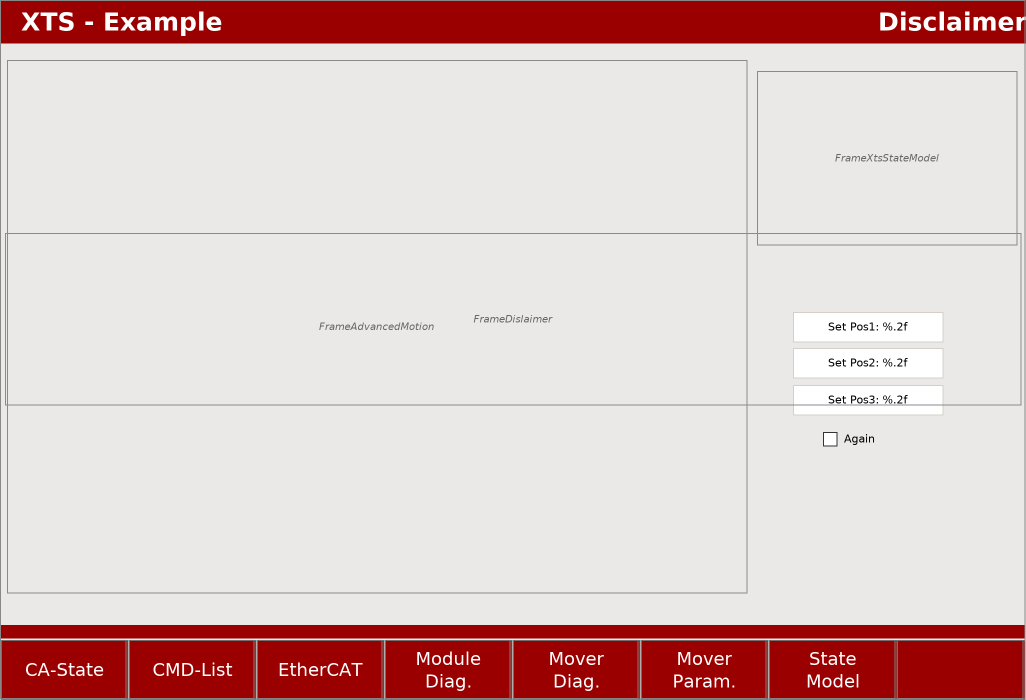
VISUALIZATION FrameVisuSimpelCaExample  // 1026x700
VAR_IN_OUT
	
	stVisuIO		: ST_VisuExampleIO;


	
END_VAR

VAR
	sVisuXtsDiag		: STRING := 'Visu_XtsDiag';
	nFrameSelect		: INT;
	
	bShowDisclaimer		: BOOL;
END_VAR
    Rectangle (1,0 1024x43), "XTS - Example"
    Rectangle (1,625 1024x13)
    Button (1,640 127x60), "CA-State", input disabled if: nFrameSelect = 0
        OnMouseClick: execute { nFrameSelect := 0; }
    Button (129,640 127x60), "CMD-List", input disabled if: (nFrameSelect = 1) or true
        OnMouseClick: execute { nFrameSelect := 1; }
    Button (257,640 127x60), "EtherCAT", input disabled if: (nFrameSelect =2) or true
        OnMouseClick: execute { nFrameSelect := 2; }
    Button (385,640 127x60), "Module Diag.", input disabled if: (nFrameSelect = 3) or true
        OnMouseClick: execute { nFrameSelect := 3; }
    Button (513,640 127x60), "Mover Diag.", input disabled if: (nFrameSelect = 4) or true
        OnMouseClick: execute { nFrameSelect := 4; }
    Button (641,640 127x60), "Mover Param.", input disabled if: (nFrameSelect = 5) or true
        OnMouseClick: execute { nFrameSelect := 5; }
    Button (897,640 128x60)
    Button (769,640 128x60), "State Model", input disabled if: nFrameSelect = 6
        OnMouseClick: execute { nFrameSelect:= 6; }
    Textfield (793,312 150x30), "Set Pos1: %.2f", text variable: stVisuIO.fSetPos1
        OnMouseClick: write the text variable via Default, min 0, max 50000
    Textfield (793,348 150x30), "Set Pos2: %.2f", text variable: stVisuIO.fSetPos2
        OnMouseClick: write the text variable via Default, min 0, max 50000
    Checkbox (821,424 94x30), "Again", variable: stVisuIO.bAgain
    Textfield (793,385 150x30), "Set Pos3: %.2f", text variable: stVisuIO.fSetPos3
        OnMouseClick: write the text variable via Default, min 0, max 50000
    Frame (7,60 740x533), frame switch variable: nFrameSelect
        shows FrameAdvancedMotion(stCaGroup := stVisuIO.stCaGroup)
        shows FrameDummy()
        shows FrameDummy()
        shows FrameDummy()
        shows FrameDummy()
        shows FrameDummy()
        shows FrameXtsStateModel(eOPMState := stVisuIO.eOPMState, eStateCommand := stVisuIO.eStateCommand)
    Frame (757,71 260x174), frame switch variable: nFrameSelect
        shows FrameXtsStateModel(eOPMState := stVisuIO.eOPMState, eStateCommand := stVisuIO.eStateCommand)
        shows FrameXtsStateModel(eOPMState := stVisuIO.eOPMState, eStateCommand := stVisuIO.eStateCommand)
        shows FrameXtsStateModel(eOPMState := stVisuIO.eOPMState, eStateCommand := stVisuIO.eStateCommand)
        shows FrameXtsStateModel(eOPMState := stVisuIO.eOPMState, eStateCommand := stVisuIO.eStateCommand)
        shows FrameXtsStateModel(eOPMState := stVisuIO.eOPMState, eStateCommand := stVisuIO.eStateCommand)
        shows FrameXtsStateModel(eOPMState := stVisuIO.eOPMState, eStateCommand := stVisuIO.eStateCommand)
        shows FrameAdvancedMotion(stCaGroup := stVisuIO.stCaGroup)
    Rectangle (875,0 151x43), "Disclaimer"
        toggle bShowDisclaimer
    Frame (5,233 1016x172), invisible if: not bShowDisclaimer
        shows FrameDislaimer()
END_VISUALIZATION

(* stored: Version 1.1.0.1, ProductVersion 3.1.4024.12
   Visu FrameVisuSimpelCaExample: Id {f1e06078-b875-44d9-89f3-dfcb5446d27a} *)
